FUNCTION_BLOCK FB_DEBOUNCE
VAR_INPUT
	SignalIn		: BOOL;
	DebounceDelay	: TIME;
END_VAR
VAR_OUTPUT
	SignalOut		: BOOL;
END_VAR
VAR
	DebounceTimer	: TON;
END_VAR



DebounceTimer.PT := DebounceDelay;

IF SignalIn <> SignalOut THEN
	DebounceTimer.IN := TRUE;
	IF DebounceTimer.Q THEN
		SignalOut := SignalIn;
		DebounceTimer.IN := FALSE;
	END_IF
ELSE
	DebounceTimer.IN := FALSE;
END_IF

DebounceTimer();

END_FUNCTION_BLOCK

(* stored: Version 1.1.0.1, ProductVersion 3.1.4024.12
   POU FB_DEBOUNCE: Id {c54d3cae-6ffa-4c99-87fd-200976859ebd}, SpecialFunc None *)
